{attribute 'GeneratedUsingTerminal: EL3773-0000-0021'}
{attribute addProperty BoxType "EL3773-0000-0021"}
{attribute addProperty Id "Sample_CountAT %I*UINT2"}
{attribute addProperty CRC "3934833369"}
{attribute addProperty Size "2"}
TYPE AI_Sample_Count_EA88CAD9 EXTENDS TcoIo.InputBase_8311D824 :
STRUCT
	{attribute addProperty Name "Sample_Count"}
	Sample_Count AT %I* : UINT;
END_STRUCT
END_TYPE

(* stored: Version 1.2.0.0, ProductVersion 3.1.4024.11
   DUT AI_Sample_Count_EA88CAD9: Id {c7bad5c7-7c0f-069c-26fc-e3e3fdd5c019} *)
